// TIA Portal V18 export
// export: Created 2025-12-01T17:53:04.1320706Z, ExportSetting None, DisplayName Totally Integrated Automation Portal, DisplayVersion V18 Update 5, DisplayName TIA Portal Openness, DisplayVersion V18 Update 5, DisplayName TIA Portal Teamcenter Gateway, DisplayVersion V18, DisplayName TIA Portal Version Control Interface, DisplayVersion V18, DisplayName STEP 7 Professional, DisplayVersion V18 Update 5, DisplayName STEP 7 Safety, DisplayVersion V18, DisplayName WinCC Professional, DisplayVersion V18 Update 5
Screen "267_Motor_H3"  1280x800, Number=267, Template=02ManualUnit1
  ScreenLayer "Layer_0"
    Button "btnMenu6_1" at 768,725 size 128x75  TextOff="H-电机3 / H-气缸3", TextOn="H-电机3 / H-气缸3"
      on Click: ActivateScreen(Screen name := , Object number := 0)
    FaceplateInstance "Motor_1" at 70,138 size 273x159  FaceplateTypeName=03 FunctionBlocks@$@202 Conveyer_Line@$@202.2 HMI@$@Motor V 0.0.7
      MotorControl := MotorControl_Dev{1}
      InterfacePropertyText "TextName"  Text="H_提升电机 / H_Lifting Motor"
    FaceplateInstance "Motor_2" at 370,138 size 273x159  FaceplateTypeName=03 FunctionBlocks@$@202 Conveyer_Line@$@202.2 HMI@$@Motor V 0.0.7
      MotorControl := MotorControl_Dev{11}
      InterfacePropertyText "TextName"  Text="H_Shaft上料电机 / H_ShaftLoadingMotor / H流线电机"
    FaceplateInstance "Motor_3" at 670,138 size 273x159  FaceplateTypeName=03 FunctionBlocks@$@202 Conveyer_Line@$@202.2 HMI@$@Motor V 0.0.7
      MotorControl := MotorControl_Dev{12}
      InterfacePropertyText "TextName"  Text="H_haft下料电机 / H_ShaftTakeMotor / H流线电机"
    Button "按钮_9" at 128,725 size 128x75  PictureOff=向右箭头_0, TextOff="H-气缸1 / H-Cylinder1", TextOn="H-气缸1 / H-Cylinder1"
      on Click: ActivateScreen(Screen name := 260_Cylinder_H1, Object number := 0)
    Button "btnMenu4" at 384,725 size 128x75  TextOff="H-气缸2 / H-Cylinder2", TextOn="H-气缸2 / H-Cylinder2"
      on Click: ActivateScreen(Screen name := 263_Cylinder_H2, Object number := 0)
    Button "btnMenu5" at 512,725 size 128x75  TextOff="H-电机2 / H-Motor2", TextOn="H-电机2 / H-Motor2"
      on Click: ActivateScreen(Screen name := 264_Motor_H2, Object number := 0)
    Button "btnMenu6" at 640,725 size 128x75  TextOff="H-气缸3 / H-Cylinder3", TextOn="H-气缸3 / H-Cylinder3"
      on Click: ActivateScreen(Screen name := 266_Cylinder_H3, Object number := 0)
    Button "btnMenu7" at 896,725 size 128x75
    Button "btnMenu7_1" at 1024,725 size 128x75
    Button "btnMenu4_1" at 256,725 size 128x75  TextOff="H-电机1 / H-Motor1", TextOn="H-电机1 / H-Motor1"
      on Click: ActivateScreen(Screen name := 261_Motor_H1, Object number := 0)
